(*~
	<docu>
		<summary>
		 	 <see cref="MatrixAccessor">See Matrix accessor</see>
			 Allows access to the elements of the parent matrix as if it were transposed
		</summary>			
	</docu>
~*)
FUNCTION_BLOCK TransposeMatrixAccessor EXTENDS MatrixAccessor
VAR_INPUT
END_VAR
VAR_OUTPUT
END_VAR
VAR
	RowRemoved_ : UINT;
	ColRemoved_ : UINT;
END_VAR

(*~
<docu>
	<inheritdoc/>			
</docu>
~*)
PROPERTY PUBLIC Cols : UINT
GET
IF NOT __ISVALIDREF(M_) THEN
	Cols := 0;
	LogWarning('%s Attempted Cols access using uninitialized Matrix Accessor');
ELSE
	Cols := M_.Rows;
END_IF
END_GET
END_PROPERTY

METHOD PUBLIC Init
VAR_INPUT
	M : REFERENCE TO Matrix;
END_VAR
Init_(M);
END_METHOD

(*~
	<docu>
		<inheritdoc/>			
	</docu>
~*)
PROPERTY PUBLIC Rows : UINT
GET
IF NOT __ISVALIDREF(M_) THEN
	Rows := 0;
	LogWarning('%s Attempted Rows access using uninitialized Matrix Accessor');
ELSE
	Rows := M_.Cols;
END_IF
END_GET
END_PROPERTY

METHOD PROTECTED This2Parent : UINT
VAR_INPUT
	Index : UINT;
END_VAR
VAR
	ThisR : UINT;
	ThisC : UINT;
END_VAR
IF NOT __ISVALIDREF(M_) THEN
	LogWarning('%s Attempted This2Parent calculation using uninitialized Matrix Accessor');
	This2Parent := 0;
	RETURN;
END_IF

IC2RC(Index,Cols,Row => ThisR, Col => ThisC);

This2Parent := RCC2I(ThisC,ThisR,M_.Cols);
END_METHOD

END_FUNCTION_BLOCK

(* stored: Version 1.1.0.1, ProductVersion 3.1.4024.9
   POU TransposeMatrixAccessor: Id {9a28d6e8-49de-0d4d-265c-dd2a9870f8ee}, SpecialFunc None
   Folder Initializers: Id {7c0114cd-41d1-0d49-1cd5-8a0554f73bcf}
   Folder Overrides: Id {c3ed05e4-8f1f-022e-21ba-86d9c4d0a320}
   Property Cols: Id {bf0da9f9-be70-0115-3902-7943e66150d7}
   Get Get: Id {cb7fdd63-8d83-06fd-2e61-15e9782a8d8f}
   Method Init: Id {cce5b477-a9bd-0f97-0e9c-4e49f12ee13b}
   Property Rows: Id {5191cf39-179d-048b-094b-53b45da5d542}
   Get Get: Id {f7be0edf-342d-0112-1abb-ce9cd40f7cf7}
   Method This2Parent: Id {82b9f386-d002-0cf1-1dd5-3226c42f62b8} *)
